{attribute 'linkalways'} 
{attribute 'no_explicit_call' := 'This FB is a CLASS and must be accessed using methods or properties'}
{attribute 'enable_dynamic_creation'}
FUNCTION_BLOCK _Array0to3OfUINT EXTENDS ArrayDatatypeBase
VAR CONSTANT
	lBound : DINT := 0;
	uBound : DINT := 3;
END_VAR
VAR
	localData : ARRAY [lBound..uBound] OF UINT;
	activeData : REFERENCE TO ARRAY [lBound..uBound] OF UINT REF= localData;
	elements : ARRAY [lBound..uBound] OF _UINT(0);
	baseType : _UINT(0);
END_VAR

PROPERTY PUBLIC Address : PVOID
GET
Address := ADR(activeData);
END_GET
END_PROPERTY

PROPERTY PUBLIC BaseDatatype : I_Datatype
GET
BaseDatatype := baseType;
END_GET
END_PROPERTY

METHOD PUBLIC ClearReference
VAR_INPUT
END_VAR
activeData REF= localData;
SetElementReference();
END_METHOD

METHOD PUBLIC Clone : I_Datatype
VAR
    pClone : POINTER TO _Array0to3OfUINT;
END_VAR
pClone := __NEW(_Array0to3OfUINT());
pClone^.Value := Value;
Clone := pClone^;
END_METHOD

METHOD FB_init : BOOL
VAR_INPUT
	bInitRetains : BOOL; // if TRUE, the retain variables are initialized (warm start / cold start)
	bInCopyCode : BOOL;  // if TRUE, the instance afterwards gets moved into the copy code (online change)
END_VAR
SetElementReference();
END_METHOD

METHOD PUBLIC GetElementAsDatatypeByIndex : I_Datatype
VAR_INPUT
	Index : DINT;
END_VAR
GetElementAsDatatypeByIndex := elements[Index];
END_METHOD

METHOD PUBLIC GetElementByIndex : REFERENCE TO _UINT;
VAR_INPUT
	Index : DINT;
END_VAR
GetElementByIndex REF= elements[Index];
END_METHOD

PROPERTY PUBLIC LowerBound : DINT
GET
LowerBound := lBound;
END_GET
END_PROPERTY

METHOD PUBLIC MakeReferenceTo
VAR_INPUT
	ReferenceTarget : REFERENCE TO ARRAY [lBound..uBound] OF UINT;
END_VAR
activeData REF= ReferenceTarget;
SetElementReference();
END_METHOD

METHOD PROTECTED OnSerializeArrayValues
VAR_INPUT
	Serializer : I_Serializer;
END_VAR
VAR
	i : DINT;
END_VAR
FOR i := lBound TO uBound DO
	elements[i].SerializeWith(Serializer);
END_FOR
END_METHOD

METHOD PROTECTED SetElementReference
VAR_INPUT
END_VAR
VAR
	i : DINT;
END_VAR
FOR i := lBound TO uBound DO
	elements[i].MakeReferenceTo(activeData[i]);
END_FOR
END_METHOD

PROPERTY PUBLIC Size : UDINT
GET
Size := SIZEOF(activeData);
END_GET
END_PROPERTY

METHOD PROTECTED TryDeserializeArrayValues : BOOL
VAR_INPUT
	Deserializer : I_Deserializer;
	Feedback : I_DeserializerFeedback;
END_VAR
VAR
	enumerator : I_DeserializerArrayForwardEnumerator;
	i : DINT;
END_VAR
enumerator := Deserializer.GetArrayEnumerator();
i := lBound;

WHILE enumerator.MoveNext() AND i <= uBound DO
	
	IF NOT elements[i].TryDeserializeFrom(enumerator.Current, Feedback) THEN
		EXIT;
	END_IF
	i := i + 1;

END_WHILE
enumerator.Dispose();
END_METHOD

METHOD TryMakeReferenceTo : BOOL
VAR_INPUT
	Target : I_Datatype;
END_VAR
VAR
	targetAsArray : I_ArrayDatatype;
	pTargetData : POINTER TO ARRAY [lBound..uBound] OF UINT;
END_VAR
IF NOT Target.TryResolveAsArrayDatatype(targetAsArray) THEN
	RETURN;
END_IF

IF NOT (targetAsArray.Identifier = Identifier) THEN
	RETURN;
END_IF

pTargetData := Target.Address;
activeData REF= pTargetData^;
SetElementReference();
TryMakeReferenceTo := TRUE;
END_METHOD

PROPERTY PUBLIC UpperBound : DINT
GET
UpperBound := ubound;
END_GET
END_PROPERTY

PROPERTY PUBLIC Value : REFERENCE TO ARRAY [lBound..uBound] OF UINT;
GET
Value ref= activeData;
END_GET
END_PROPERTY

END_FUNCTION_BLOCK

(* stored: Version 1.1.0.1, ProductVersion 3.1.4024.13
   POU _Array0to3OfUINT: Id {c3a26628-c459-031d-33a9-3fffa547078d}, SpecialFunc None
   Folder Core: Id {eb0356bb-342e-0569-0691-c9d2a5747038}
   Folder Constructor: Id {c3110e1d-3f45-08d5-38d9-cb5bdf76b4c3}
   Folder Protected: Id {0c875e4f-6d80-0c89-0e26-19a3032a6c04}
   Folder Customize: Id {59191baf-95ed-0bf6-1c02-12e0bdd076a3}
   Property Address: Id {78f79bc2-2d0f-0d31-07cd-f19a23dd8fa6}
   Get Get: Id {7633efa1-223b-02ec-0012-e0877044230b}
   Property BaseDatatype: Id {be332cf2-58fe-0b69-370c-03b871ffe860}
   Get Get: Id {595010f8-ca03-0663-0407-5559e7d5130e}
   Method ClearReference: Id {f4bf6353-6974-0673-1da5-5078a5427264}
   Method Clone: Id {663d0f86-5953-05db-2ad4-b2f2ae96e4b2}
   Method FB_init: Id {52258580-5191-0fca-2f09-76c6812b34a3}
   Method GetElementAsDatatypeByIndex: Id {520cc8ac-ea26-0ac2-2944-76bb12374260}
   Method GetElementByIndex: Id {fa626b1c-894d-004f-20a8-d00606efea79}
   Property LowerBound: Id {85ff1c1a-98c5-054d-2c74-00bcd38b5d7b}
   Get Get: Id {0e5f9096-819c-0ab3-371d-9c4f8ea37014}
   Method MakeReferenceTo: Id {4489b418-9725-0a0e-07b9-2e904ac3cecf}
   Method OnSerializeArrayValues: Id {7cae1342-1d63-05e6-033c-103c2feef2b0}
   Method SetElementReference: Id {dd3d1713-72db-0d5f-14fb-37f6f4446ad0}
   Property Size: Id {e4a4da99-938b-0ad6-2d07-e717d718769a}
   Get Get: Id {e615d9e9-ffd4-06af-049e-ccf0ba50357d}
   Method TryDeserializeArrayValues: Id {4f62e0a9-64c8-06b7-2a80-50d955cf9d25}
   Method TryMakeReferenceTo: Id {0092f664-e65c-0a74-2acd-19af5fed976b}
   Property UpperBound: Id {448704b6-738e-0a13-2a2d-c272d84769a2}
   Get Get: Id {b14ff36a-8e34-0c85-33a6-947a69613583}
   Property Value: Id {8b19877f-4ed5-0583-23d0-d8b9fd791b7d}
   Get Get: Id {7ba79c2c-f684-0e75-10de-ea6c9a45153f} *)
